// TIA Portal V17 export
// export: Created 2023-12-22T15:05:35.8671424Z, ExportSetting WithDefaults, DisplayName Totally Integrated Automation Portal, DisplayVersion V17, DisplayName TIA Portal Openness, DisplayVersion V17, DisplayName TIA Portal Version Control Interface, DisplayVersion V17, DisplayName STEP 7 Professional, DisplayVersion V17, DisplayName STEP 7 Safety, DisplayVersion V17, DisplayName WinCC Advanced, DisplayVersion V17
TYPE "PolyMix_Report"
// stored: IsFailsafeCompliant false
   STRUCT
      C : Real;   // Средняя концентрация
      Water : Real;   // Расход воды, литры
      Reagent : Real;   // Расход реагента по дозатору, кг
      Weight : Real;   // Расход реагента по весам, кг
      Dos : Real;   // Число доз
      Res : Real;   // Наработка, часы
      WeekDay : Int;   // День недели
      Day : Int;   // Дата записи
      Month : Int;   // Месяц записи
   END_STRUCT;
END_TYPE
